FUNCTION TwoPiCrop : REAL
VAR_INPUT
	in:REAL;
END_VAR
VAR
	aux_LINT:LINT;
END_VAR

aux_LINT:=REAL_TO_LINT(in*1000000);
aux_LINT:= aux_LINT MOD REAL_TO_LINT(1000000*2*GVL.Pi);
TwoPiCrop:= LINT_TO_REAL(aux_LINT)/1000000;
IF TwoPiCrop < 0 THEN
	TwoPiCrop := 2*GVL.Pi - TwoPiCrop;
END_IF

END_FUNCTION

(* stored: Version 1.1.0.1, ProductVersion 3.1.4024.4
   POU TwoPiCrop: Id {65dcc3c2-f5ba-43ee-ac6a-141ce6fc5669}, SpecialFunc None *)
